FUNCTION_BLOCK TFCiclo_Deposito_Falda
VAR_INPUT
	Ciclo 		: POINTER TO Stato_Ciclo_Lavoro;
	Programma  : POINTER TO TFProgramma_Ciclo_Falda_Lastre;
	ModuleAX_X : POINTER TO TFModulePalletizer_Ax;
	ModuleAX_Y : POINTER TO TFModulePalletizer_Ax;
	ModuleAX_Z : POINTER TO TFModulePalletizer_Ax;
	ModuleAX_J : POINTER TO TFModulePalletizer_AxJ_Lastre;
	StartInterpolazioneAssi : POINTER TO BOOL;
	QuotaPassModePuntoIntermedio : ARRAY [1..3] OF REAL;
	ModulePinza : POINTER TO TFModulePalletizer_Pinza;
	TipoDiDeposito : UINT;
	AbilitazioneGlobalePassMode	: BOOL;
	InterrompiCiclo : BOOL;
	Abilita_Ciclo_Step : BOOL;
	Command_Step : BOOL;
	AbilitazioneAnticipoDinamicoMovimenti : BOOL;
END_VAR
VAR_OUTPUT
	STEPDone	: BOOL;
END_VAR
VAR
	StepInto: BOOL;
END_VAR

(* Set della variabile che mi permette di fare lo STEP nel ciclo *)
StepInto := (Abilita_Ciclo_Step AND Command_Step) OR NOT Abilita_Ciclo_Step;

(* Reset Anticipo Dinamico se non ho l'abilitazione *)
IF NOT AbilitazioneAnticipoDinamicoMovimenti  OR NOT HMI_DisabilitaAnticipiGLOBALE THEN
	QuotaAnticipoDinamicaX_Raggiunta := FALSE;
	QuotaAnticipoDinamicaY_Raggiunta := FALSE;
	QuotaAnticipoDinamicaZ_Raggiunta := FALSE;
END_IF

IF NOT InterrompiCiclo THEN
	IF Ciclo^.Stato = TERMINATO OR Ciclo^.Stato = ANNULLATO THEN
		Ciclo^.Passo := 0;
	ELSIF Ciclo^.Stato = INTERROTTO THEN
		Ciclo^.Passo := 999;
	END_IF
	Ciclo^.Stato := IN_ESECUZIONE;
	CASE Ciclo^.Passo OF
	(* Case 0 *)
			0:  Ciclo^.Stato := IN_ESECUZIONE;
				Ciclo^.Passo := 10;
				STEPDone := FALSE;
		
			(* Case 10 - PROGRAMMA[53] ASSE Z -> TRASLAZIONE A QUOTA DI "ATTESA CADUTA FALDA" *)	
			10:	
				Ciclo^.Stato := IN_ESECUZIONE;
				IF StepInto THEN
					Programma_Z[53].Stato := DA_ESEGUIRE;
					Programma_Z[53].InterpolaAsse := NO_INTERPOLAZIONE_ASSE;//FALSE;//NO_INTERPOLAZIONE_ASSE
					ProgrammaToModule_Z := Programma_Z[53];
					Ciclo^.Passo := 11;
					STEPDone := FALSE;
				END_IF
				
			(* Case 11 - Attesa completamento del comando MOVETOPOS o del raggiungimento quota di Pre-Movimento se abilitata la funzione*)
			11: 
				IF Programma_Z[53].Stato = TERMINATO OR
				(ModuleAX_Z^.Ax^.Status.ActPosition >= Programma^.Quota_Attesa_Caduta_Falda_Z - 50) THEN // con -30 faccio in modo che il programma successivo si innesti a quello in corso.. per non vedere lo stacco...
					Ciclo^.Passo := 20;
					STEPDone := TRUE;
				ELSIF Programma_Z[53].Stato = INTERROTTO THEN
					Ciclo^.Passo := 10;										
				END_IF
				
			(* Case 20 - PROGRAMMA[54] ASSE Z -> TRASLAZIONE A QUOTA DI FUORI INGOMBRO *)	
			20:	Ciclo^.Stato := IN_ESECUZIONE;
				IF StepInto THEN
					Programma_Z[54].Stato := DA_ESEGUIRE;
					Programma_Z[54].InterpolaAsse := NO_INTERPOLAZIONE_ASSE;//FALSE;//NO_INTERPOLAZIONE_ASSE
					ProgrammaToModule_Z := Programma_Z[54];
					Ciclo^.Passo := 21;
					STEPDone := FALSE;
				END_IF
				
			(* Case 21 - Attesa completamento del comando MOVETOPOS o del raggiungimento quota di Pre-Movimento se abilitata la funzione *)
			21: 
				IF Programma_Z[54].Stato = TERMINATO OR
					(ModuleAX_Z^.Ax^.Status.ActPosition >= QuotaFuoriIngombro_Z_ConFALDA) OR 
					(Asse_Z_InFinestraDiPassMode AND Programma_Z[54].Stato = IN_ESECUZIONE) THEN
						IF (TipoDiDeposito = DEPOSITO_FALDA_SU_CATASTA AND ((Mission.PPick-1)=Mission.PPlace)) THEN//Vado direttamente in prelievo senza fare il fuori ingombro SE devo depositare sulla catasta e la catasta è di fronte al mag. falde 
							Ciclo^.Passo := 40;
							STEPDone := TRUE;
						ELSE
							Ciclo^.Passo := 22;
							STEPDone := TRUE;
						END_IF
				ELSIF Programma_Z[54].Stato = INTERROTTO THEN
					Ciclo^.Passo := 20;										
				END_IF
				
			(* Case 22 - Vado a quota di fuori ingombro colonne con Y *)
			22:
				IF Programma_Z[54].Stato = INTERROTTO THEN
					 Ciclo^.Passo := 20;										
				ELSE
					IF StepInto THEN
						Programma_Y[66].Stato := DA_ESEGUIRE;
						Programma_Y[66].InterpolaAsse := NO_INTERPOLAZIONE_ASSE;
						ProgrammaToModule_Y := Programma_Y[66];
						Ciclo^.Passo := 23;
						STEPDone := FALSE;
					END_IF
				END_IF
					
			(* Case 23 - Arrivato a quota di fuori ingombro colonne con Y *)		
			23:
				IF Programma_Z[54].Stato = INTERROTTO OR 
					Programma_Y[66].Stato = INTERROTTO THEN
						Ciclo^.Passo := 20;
				ELSE	
					IF Programma_Y[66].Stato = TERMINATO OR Asse_Y_InFinestraDiPassMode THEN
						Ciclo^.Passo := 40;
						STEPDone := TRUE;							
					END_IF
				END_IF
				
			(* Case 40 - PROGRAMMA[..] ASSE  -> TRASLAZIONE A QUOTA DI DEPOSITO FALDA  *)	
			40:	
				IF Programma_Z[54].Stato = INTERROTTO THEN					
					Ciclo^.Passo := 20;										
				ELSE
					IF TipoDiDeposito = DEPOSITO_FALDA_SU_CATASTA THEN
						IF StepInto THEN
							Programma_X[52].Stato := DA_ESEGUIRE;
							Programma_X[52].InterpolaAsse := INTERPOLAZIONE_ASSE;//TRUE;//INTERPOLAZIONE_ASSE
							ProgrammaToModule_X := Programma_X[52];
							IF NOT Pinza_InIngombroColonne_Destinazione THEN
								Programma_Y[52].Stato := DA_ESEGUIRE;
								Programma_Y[52].InterpolaAsse := INTERPOLAZIONE_ASSE;//TRUE;//INTERPOLAZIONE_ASSE
								ProgrammaToModule_Y := Programma_Y[52];
							END_IF
							Programma_J[11].Stato := DA_ESEGUIRE;
							Programma_J[11].InterpolaAsse := INTERPOLAZIONE_ASSE;//TRUE;//INTERPOLAZIONE_ASSE
							ProgrammaToModule_J := Programma_J[11];
							
							Programma_K[53].Stato := DA_ESEGUIRE;
							Programma_K[53].InterpolaAsse := NO_INTERPOLAZIONE_ASSE;//FALSE;//NO_INTERPOLAZIONE_ASSE
							ProgrammaToModule_K := Programma_K[53];
							
							ProgrammaToModule_Z.InterpolaAsse := NO_INTERPOLAZIONE_ASSE;//FALSE;
							
							StartInterpolazioneAssi^ := TRUE; //Abilito l'interpolazione degli assi

							Ciclo^.Passo := 41;
							STEPDone := FALSE;
						END_IF
					ELSIF TipoDiDeposito = DEPOSITO_FALDA_SU_PIAZZOLA THEN
						IF StepInto THEN
							Programma_X[53].Stato := DA_ESEGUIRE;
							Programma_X[53].InterpolaAsse := INTERPOLAZIONE_ASSE;//TRUE;//INTERPOLAZIONE_ASSE
							ProgrammaToModule_X := Programma_X[53];
							(*IF NOT Pinza_InIngombroColonne_Destinazione THEN
								Programma_Y[53].Stato := DA_ESEGUIRE;
								Programma_Y[53].InterpolaAsse := INTERPOLAZIONE_ASSE;//TRUE;//INTERPOLAZIONE_ASSE
								ProgrammaToModule_Y := Programma_Y[53];
							END_IF*)
							Programma_J[11].Stato := DA_ESEGUIRE;
							Programma_J[11].InterpolaAsse := INTERPOLAZIONE_ASSE;//TRUE;//INTERPOLAZIONE_ASSE
							ProgrammaToModule_J := Programma_J[11];
							
							Programma_K[53].Stato := DA_ESEGUIRE;
							Programma_K[53].InterpolaAsse := NO_INTERPOLAZIONE_ASSE;//FALSE;//NO_INTERPOLAZIONE_ASSE
							ProgrammaToModule_K := Programma_K[53];
							
							StartInterpolazioneAssi^ := TRUE; //Abilito l'interpolazione degli assi							
						
							Ciclo^.Passo := 41;
							STEPDone := FALSE;
						END_IF
					ELSE
						;
					END_IF
				END_IF
			
			41: IF Programma_Z[54].Stato = INTERROTTO THEN					
					Ciclo^.Passo := 20;										
				ELSE
					STEPDone := TRUE;
					IF QuotaX_ConsensoRotazionePinza_Raggiunta OR NOT Pinza_InIngombroColonne_Destinazione THEN
						IF TipoDiDeposito = DEPOSITO_FALDA_SU_CATASTA THEN
							IF StepInto THEN
								Programma_Y[52].Stato := DA_ESEGUIRE;
								Programma_Y[52].InterpolaAsse := NO_INTERPOLAZIONE_ASSE;//TRUE;//INTERPOLAZIONE_ASSE
								ProgrammaToModule_Y := Programma_Y[52];
								
								Ciclo^.Passo := 42;
								STEPDone := FALSE;
							END_IF
						ELSIF TipoDiDeposito = DEPOSITO_FALDA_SU_PIAZZOLA THEN
							IF StepInto THEN
								Programma_Y[53].Stato := DA_ESEGUIRE;
								Programma_Y[53].InterpolaAsse := NO_INTERPOLAZIONE_ASSE;//TRUE;//INTERPOLAZIONE_ASSE
								ProgrammaToModule_Y := Programma_Y[53];
								
								Ciclo^.Passo := 42;
								STEPDone := FALSE;
							END_IF
						ELSE
							;
						END_IF
					END_IF
				END_IF	
						
			(* Case 42 -  Attesa completamento del comando MOVETOPOS o del raggiungimento quota di Pre-Movimento se abilitata la funzione *)
			42: 
				IF Programma_Z[54].Stato = INTERROTTO OR 
					(TipoDiDeposito = DEPOSITO_FALDA_SU_CATASTA AND Programma_X[52].Stato = INTERROTTO) OR 
					(TipoDiDeposito = DEPOSITO_FALDA_SU_PIAZZOLA AND Programma_X[53].Stato = INTERROTTO) OR
					(TipoDiDeposito = DEPOSITO_FALDA_SU_CATASTA  AND Programma_Y[52].Stato = INTERROTTO) OR
					(TipoDiDeposito = DEPOSITO_FALDA_SU_PIAZZOLA AND Programma_Y[53].Stato = INTERROTTO) OR
					Programma_J[11].Stato = INTERROTTO OR
					Programma_K[53].Stato = INTERROTTO THEN
						Ciclo^.Passo := 20;	
				(* Deposito su catasta *)
				ELSIF TipoDiDeposito = DEPOSITO_FALDA_SU_CATASTA THEN
					IF (Programma_X[52].Stato = TERMINATO OR Asse_X_InFinestraDiPassMode) AND
						(Programma_Y[52].Stato = TERMINATO OR Asse_Y_InFinestraDiPassMode) AND  
					  	Programma_J[11].Stato = TERMINATO AND 
						Programma_K[53].Stato = TERMINATO THEN 
							Ciclo^.Passo := 50;
							STEPDone := TRUE;
					END_IF
				(* Deposito Su piazzola *)
				ELSIF (Programma_X[53].Stato = TERMINATO OR Asse_X_InFinestraDiPassMode) AND 
					  (Programma_Y[53].Stato = TERMINATO OR Asse_Y_InFinestraDiPassMode) AND
					  Programma_J[11].Stato = TERMINATO AND
					  Programma_K[53].Stato = TERMINATO THEN 
							Ciclo^.Passo := 50;
							STEPDone := TRUE;								
				END_IF	
							
			(* Case 80 - PROGRAMMA[..] ASSE Z -> TRASLAZIONE A QUOTA AMMESSA IN VELOCE DI DEPOSITO FALDA  
			- DEPOSITO_FALDA_SU_CATASTA : PROGRAMMA[55] ASSE Z
			- DEPOSITO_FALDA_SU_PIAZZOLA : PROGRAMMA[57] ASSE Z *)
			50:
				IF TipoDiDeposito = DEPOSITO_FALDA_SU_CATASTA THEN
					IF StepInto THEN
						Programma_Z[55].Stato := DA_ESEGUIRE;
						Programma_Z[55].InterpolaAsse := NO_INTERPOLAZIONE_ASSE;//FALSE;//NO_INTERPOLAZIONE_ASSE
						ProgrammaToModule_Z := Programma_Z[55];
						Ciclo^.Passo := 52;
						STEPDone := FALSE;
					END_IF
				ELSIF TipoDiDeposito = DEPOSITO_FALDA_SU_PIAZZOLA THEN
					IF StepInto THEN
						Programma_Z[57].Stato := DA_ESEGUIRE;
						Programma_Z[57].InterpolaAsse := NO_INTERPOLAZIONE_ASSE;//FALSE;//NO_INTERPOLAZIONE_ASSE
						ProgrammaToModule_Z := Programma_Z[57];
						Ciclo^.Passo := 51;	//SALTO DIRETTAMENTE AL CASE 91 DOVE SI ASPETTA LA FINE DEL MOVIMENTO DELL'ASSE Z
						STEPDone := FALSE;
					END_IF
				ELSE
					;
				END_IF
					
			(* Case 51 -  Attesa completamento del comando MOVETOPOS o del raggiungimento quota di Pre-Movimento se abilitata la funzione *)
			51: 
				IF (TipoDiDeposito = DEPOSITO_FALDA_SU_CATASTA AND Programma_Z[55].Stato = INTERROTTO) OR 
				(TipoDiDeposito = DEPOSITO_FALDA_SU_PIAZZOLA AND  Programma_Z[57].Stato = INTERROTTO) THEN
					Ciclo^.Passo := 20;	//NON DOVREBBE ACCADERE									
				ELSE
					IF (TipoDiDeposito = DEPOSITO_FALDA_SU_CATASTA AND Programma_Z[55].Stato = TERMINATO) OR
					(TipoDiDeposito = DEPOSITO_FALDA_SU_PIAZZOLA AND  Programma_Z[57].Stato = TERMINATO)(*OR
						(ModuleAX_Z^.Ax^.Status.ActPosition >= TFProgramma_Ciclo_Falda.Quota_Deposito_Falda_SuPiazzola_Z)*) THEN
						Ciclo^.Passo := 110;
						STEPDone := TRUE;
					END_IF	
				END_IF
				
			(* Case 52 -  Attesa completamento del comando MOVETOPOS o del raggiungimento quota di Pre-Movimento se abilitata la funzione *)
			52: 
				IF Programma_Z[55].Stato = INTERROTTO OR Programma_Z[55].Stato = NON_ESEGUITO OR 
				(TipoDiDeposito = DEPOSITO_FALDA_SU_CATASTA AND Programma_X[52].Stato = INTERROTTO) THEN
					Ciclo^.Passo := 20;	//NON DOVREBBE ACCADERE									
				ELSE
					IF Programma_Z[55].Stato = TERMINATO OR
						(ModuleAX_Z^.Ax^.Status.ActPosition <= Programma^.Quota_StartLenta_Deposito_Falda_SuCatastaPallet_Z + 10) AND Programma_Z[56].Stato = IN_ESECUZIONE THEN
						Ciclo^.Passo := 100;
						STEPDone := TRUE;
					END_IF	
				END_IF	
				
			(* Case 100 - PROGRAMMA[56] ASSE Z -> TRASLAZIONE IN LENTA A QUOTA DI DEPOSITO FALDA SU CATASTA VUOTI  *)
			100:
				IF Programma_Z[55].Stato = INTERROTTO OR
				(TipoDiDeposito = DEPOSITO_FALDA_SU_CATASTA AND  Programma_X[52].Stato = INTERROTTO ) OR
				(TipoDiDeposito = DEPOSITO_FALDA_SU_PIAZZOLA AND (Programma_X[53].Stato = INTERROTTO OR Programma_Z[57].Stato = INTERROTTO)) THEN
					Ciclo^.Passo := 20; //NON DOVREBBE ACCADERE										
				ELSE
					IF StepInto THEN
						Programma_Z[56].Stato := DA_ESEGUIRE;
						Programma_Z[56].InterpolaAsse := NO_INTERPOLAZIONE_ASSE;//FALSE;//NO_INTERPOLAZIONE_ASSE
						ProgrammaToModule_Z := Programma_Z[56];
						Ciclo^.Passo := 101;
						STEPDone := FALSE;
					END_IF
				END_IF
			(* Case 81 -  Attesa completamento del comando MOVETOPOS o del raggiungimento quota di Pre-Movimento se abilitata la funzione *)
			101: 
				IF Programma_Z[56].Stato = INTERROTTO OR 
				(TipoDiDeposito = DEPOSITO_FALDA_SU_CATASTA 	AND NOT Programma_X[52].Stato = TERMINATO) OR
				(TipoDiDeposito = DEPOSITO_FALDA_SU_CATASTA 	AND NOT Programma_Y[52].Stato = TERMINATO) THEN
					Ciclo^.Passo := 20; //NON DOVREBBE ACCADERE										
				ELSE
					IF Programma_Z[56].Stato = TERMINATO THEN
						Ciclo^.Passo := 110;
						STEPDone := TRUE;
					END_IF	
				END_IF
				
			(* Case 110 - UNLOAD MODULO ASPIRAZIONE  *)
			110:
				IF StepInto THEN
					TFParametersArrayClear(ADR(ParametersArray));
					TFCommandSend(CmdUNLOAD,ParametersArray,ModulePinza^.Cmd);
					Ciclo^.Passo := 111;
					STEPDone := FALSE;
				END_IF

			(* Case 71 -  Attesa completamento del comando UNLOAD MODULO ASPIRAZIONE *)
			111: 
				IF TFStateCodeGet(ModulePinza^.State) = StateERROR THEN
					Ciclo^.Passo := 20;
				ELSIF NOT TFStateCodeGet(ModulePinza^.State) = StateUNLOAD_RUN  THEN
					Ciclo^.Passo := 110;										
				ELSE
					IF TFStateCodeGet(ModulePinza^.State) = StateUNLOAD_END THEN
						Ciclo^.Passo := 1000;
						STEPDone := TRUE;
					END_IF	
				END_IF

			(* Case 1000 *)
			1000:
				Ciclo^.Stato := TERMINATO;
				Ciclo^.Passo := 1000;
				
			(* Case 9999 - Ciclo NON annullato o NON terminato*)
			9999:
				Ciclo^.Stato := INTERROTTO;
				Ciclo^.Passo := 9999;
	ELSE						
		;
			
	END_CASE;
ELSE								//Se il ciclo deve essere interrotto, setto il suo nuovo stato
	Ciclo^.Stato := INTERROTTO;
END_IF

END_FUNCTION_BLOCK

(* stored: Version 1.1.0.1, ProductVersion 3.1.4024.11
   POU TFCiclo_Deposito_Falda: Id {895f47e0-98fa-438a-9511-62f6a62a887f}, SpecialFunc None *)
